% RSLogix 500 project FLASHER.RSS, saved by version 8.30.00.16 %
PROJECT "UNTITLED"    % processor: MicroLogix 1000 %

PROGRAM FILES
  LAD 2 "MAIN_PROG"  5 rungs
  LAD 3 "USER_FAULT"  1 rungs
  LAD 4 "HSC_INT"  1 rungs
  LAD 5 "STI_INT"  1 rungs
  LAD 6, 7, 8, 9, 10, 11, 12, 13, 14, 15, 16: only END

DATA FILES
  O0 OUTPUT  1 elements
  I1 INPUT  2 elements
  S2 STATUS  33 elements
  B3 BINARY  32 elements
  T4 TIMER  40 elements
  C5 COUNTER  32 elements
  R6 CONTROL  16 elements
  N7 INTEGER  105 elements

LADDER 2 "MAIN_PROG"
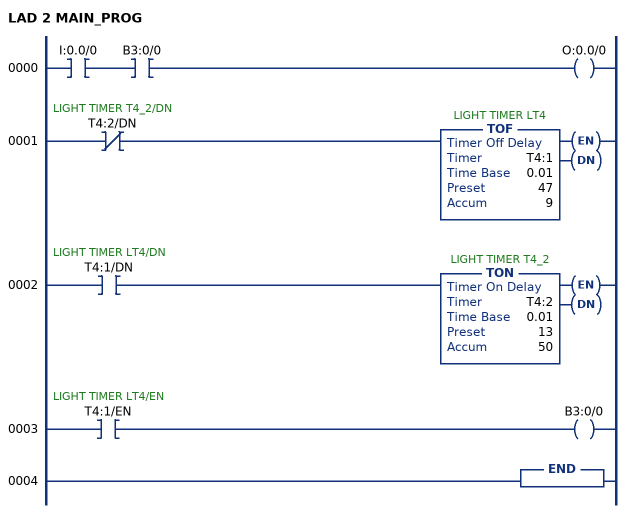
% Rung: 0 %
SOR XIC I:0.0/0 XIC B3:0/0 OTE O:0.0/0 EOR
% Rung: 1 %
SOR XIO T4:2/DN TOF T4:1 0.01 47 9 EOR
%   T4:2  T4_2  "LIGHT TIMER" %
%   T4:1  LT4  "LIGHT TIMER" %
% Rung: 2 %
SOR XIC T4:1/DN TON T4:2 0.01 13 50 EOR
%   T4:1  LT4  "LIGHT TIMER" %
%   T4:2  T4_2  "LIGHT TIMER" %
% Rung: 3 %
SOR XIC T4:1/EN OTE B3:0/0 EOR
%   T4:1  LT4  "LIGHT TIMER" %
% Rung: 4 %
SOR END EOR

OTHER DOCUMENTED ADDRESSES
  B3:0/10  FB1  "flasher bit"

DATA TABLE (non-zero values as saved)
DATA T4
% .PRE .ACC %
% T4:1 % 47 9
% T4:2 % 13 50
